// TIA Portal V19 export
FUNCTION "TimeZone" : Void   // FC4, LAD
{ S7_Optimized_Access := 'TRUE' }
// stored: SetENOAutomatically false
   VAR_IN_OUT
      Zone : "Time Zone";
   END_VAR
   VAR_TEMP
      RealTime : Time;
   END_VAR
   VAR_TEMP   // added for the SCL form of the ladder/FBD networks
      _w1 : Bool;
   END_VAR
BEGIN

REGION Network 1
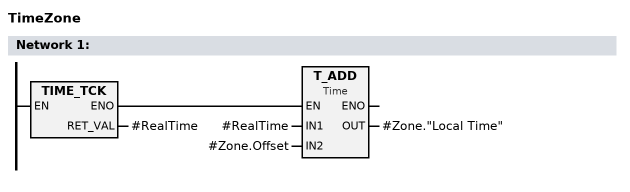
   RUNG wire#powerrail
      TIME_TCK(RET_VAL => #RealTime)
      { S7_Templates := "[date_type := Time, time_type := Time]" } T_ADD(IN1 := #RealTime, IN2 := #Zone.Offset, OUT => #Zone."Local Time")
   END_RUNG
   // the same network as SCL:
   #RealTime := TIME_TCK(ENO => #_w1);
   IF #_w1 THEN T_ADD(IN1 := #RealTime, IN2 := #Zone.Offset, OUT => #Zone."Local Time"); END_IF;
END_REGION
END_FUNCTION
